// Mitsubishi GX Developer project: Ножницы дисковые (Подольск)   PLC: FX3G

PROGRAM MAIN
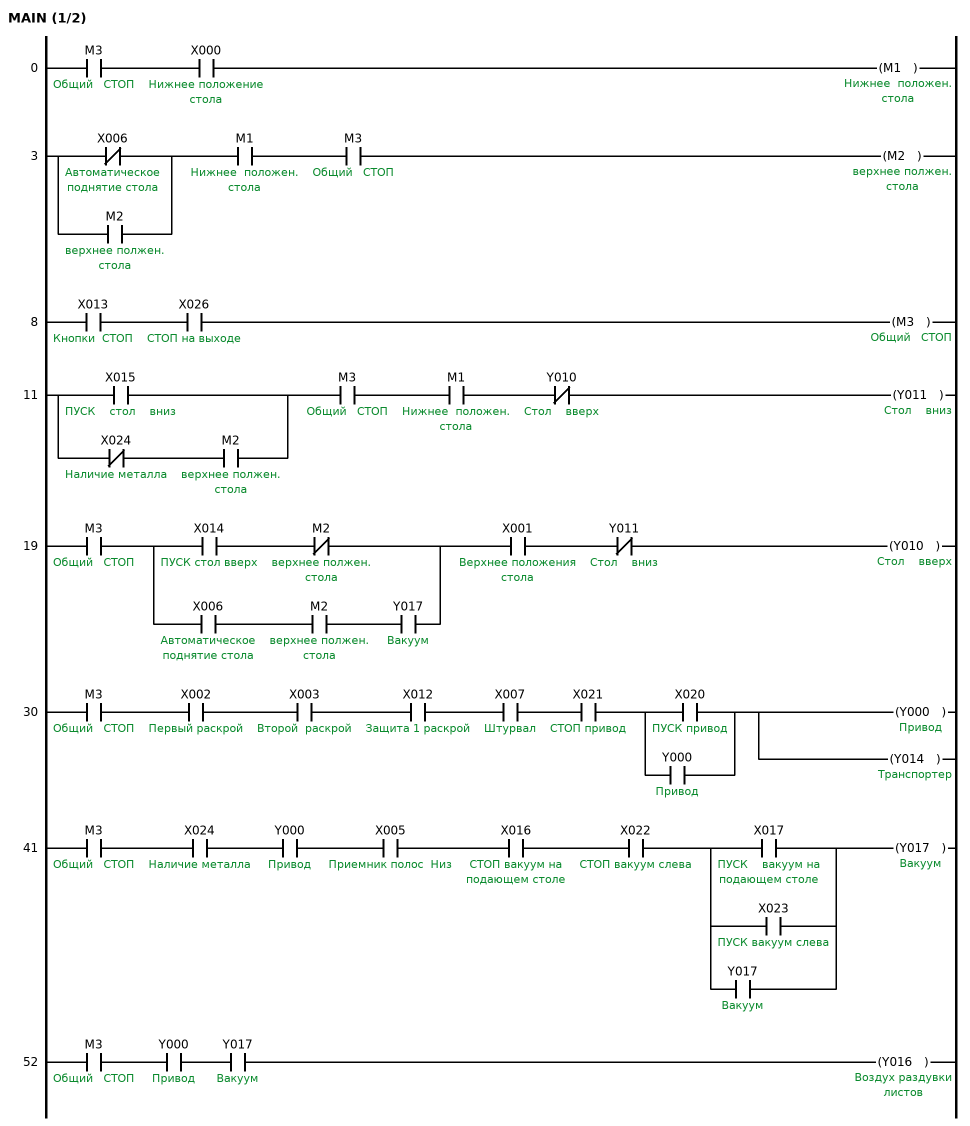
0     LD      M3  ; Общий   СТОП
      AND     X000  ; Нижнее положение стола
      OUT     M1  ; Нижнее  положен. стола
3     LDI     X006  ; Автоматическое поднятие стола
      OR      M2  ; верхнее полжен. стола
      AND     M1  ; Нижнее  положен. стола
      AND     M3  ; Общий   СТОП
      OUT     M2  ; верхнее полжен. стола
8     LD      X013  ; Кнопки  СТОП
      AND     X026  ; СТОП на выходе
      OUT     M3  ; Общий   СТОП
11    LD      X015  ; ПУСК    стол    вниз
      LDI     X024  ; Наличие металла
      AND     M2  ; верхнее полжен. стола
      ORB
      AND     M3  ; Общий   СТОП
      AND     M1  ; Нижнее  положен. стола
      ANI     Y010  ; Стол    вверх
      OUT     Y011  ; Стол    вниз
19    LD      M3  ; Общий   СТОП
      LD      X014  ; ПУСК стол вверх
      ANI     M2  ; верхнее полжен. стола
      LD      X006  ; Автоматическое поднятие стола
      AND     M2  ; верхнее полжен. стола
      AND     Y017  ; Вакуум
      ORB
      ANB
      AND     X001  ; Верхнее положения стола
      ANI     Y011  ; Стол    вниз
      OUT     Y010  ; Стол    вверх
30    LD      M3  ; Общий   СТОП
      AND     X002  ; Первый раскрой
      AND     X003  ; Второй  раскрой
      AND     X012  ; Защита 1 раскрой
      AND     X007  ; Штурвал
      AND     X021  ; СТОП привод
      LD      X020  ; ПУСК привод
      OR      Y000  ; Привод
      ANB
      OUT     Y000  ; Привод
      OUT     Y014  ; Транспортер
41    LD      M3  ; Общий   СТОП
      AND     X024  ; Наличие металла
      AND     Y000  ; Привод
      AND     X005  ; Приемник полос  Низ
      AND     X016  ; СТОП вакуум на подающем столе
      AND     X022  ; СТОП вакуум слева
      LD      X017  ; ПУСК    вакуум на подающем столе
      OR      X023  ; ПУСК вакуум слева
      OR      Y017  ; Вакуум
      ANB
      OUT     Y017  ; Вакуум
52    LD      M3  ; Общий   СТОП
      AND     Y000  ; Привод
      AND     Y017  ; Вакуум
      OUT     Y016  ; Воздух раздувки листов
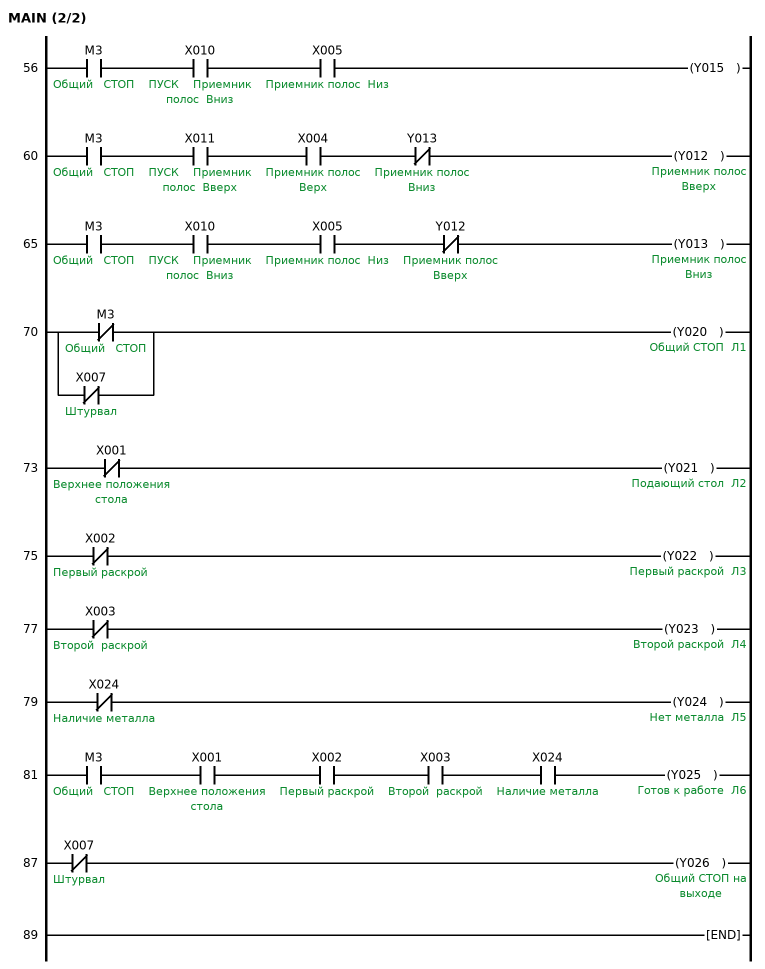
56    LD      M3  ; Общий   СТОП
      AND     X010  ; ПУСК    Приемник полос  Вниз
      AND     X005  ; Приемник полос  Низ
      OUT     Y015
60    LD      M3  ; Общий   СТОП
      AND     X011  ; ПУСК    Приемник полос  Вверх
      AND     X004  ; Приемник полос  Верх
      ANI     Y013  ; Приемник полос  Вниз
      OUT     Y012  ; Приемник полос  Вверх
65    LD      M3  ; Общий   СТОП
      AND     X010  ; ПУСК    Приемник полос  Вниз
      AND     X005  ; Приемник полос  Низ
      ANI     Y012  ; Приемник полос  Вверх
      OUT     Y013  ; Приемник полос  Вниз
70    LDI     M3  ; Общий   СТОП
      ORI     X007  ; Штурвал
      OUT     Y020  ; Общий СТОП  Л1
73    LDI     X001  ; Верхнее положения стола
      OUT     Y021  ; Подающий стол  Л2
75    LDI     X002  ; Первый раскрой
      OUT     Y022  ; Первый раскрой  Л3
77    LDI     X003  ; Второй  раскрой
      OUT     Y023  ; Второй раскрой  Л4
79    LDI     X024  ; Наличие металла
      OUT     Y024  ; Нет металла  Л5
81    LD      M3  ; Общий   СТОП
      AND     X001  ; Верхнее положения стола
      AND     X002  ; Первый раскрой
      AND     X003  ; Второй  раскрой
      AND     X024  ; Наличие металла
      OUT     Y025  ; Готов к работе  Л6
87    LDI     X007  ; Штурвал
      OUT     Y026  ; Общий СТОП на выходе
89    END
END_PROGRAM

// device comments not shown above
X025  ; Воздух раздувки
Y001  ; Привод Jog
